FUNCTION_BLOCK ARUCODETECTOR (* openCV Aruco Detector *)
  (* Version 1.0, AN, SWDC RTSoft *)
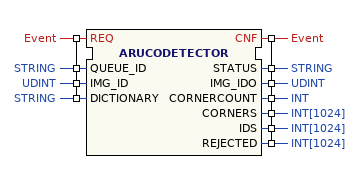
  EVENT_INPUT
    REQ WITH QUEUE_ID, IMG_ID, DICTIONARY;
  END_EVENT
  EVENT_OUTPUT
    CNF WITH STATUS, IMG_IDO, CORNERCOUNT, CORNERS, IDS, REJECTED;
  END_EVENT
  VAR_INPUT
    QUEUE_ID : STRING;
    IMG_ID : UDINT;
    DICTIONARY : STRING;
  END_VAR
  VAR_OUTPUT
    STATUS : STRING;
    IMG_IDO : UDINT;
    CORNERCOUNT : INT; (* Number of detected Aruco markers *)
    CORNERS : ARRAY [0..1023] OF INT; (* Detected Aruco marker corners *)
    IDS : ARRAY [0..1023] OF INT; (* Detected Aruco marker IDs *)
    REJECTED : ARRAY [0..1023] OF INT; (* Rejected Aruco marker candidates *)
  END_VAR
  ALGORITHM REQ IN ST:

  END_ALGORITHM
END_FUNCTION_BLOCK
